Yaskawa INFORM job: SEQUENCE1.JBI

/JOB
//NAME SEQUENCE1
//POS
///NPOS 16,16,16,0,0,0
///TOOL 2
///POSTYPE PULSE
///PULSE
C00000=-123787,24304,7596,24730,-10033,18005
C00001=-124139,38523,-23923,25034,13017,13567
C00002=-125998,37166,-27833,25904,14956,13586
C00003=-126763,36701,-29332,26274,15729,13590
C00004=-125268,29724,-35802,30017,19497,16175
C00005=-123323,21362,-43824,35562,24187,18403
C00006=-122752,14684,-49649,39024,28143,20530
C00007=-122789,12113,-51767,40794,30645,22351
C00008=-122154,60097,-5285,37527,25638,24249
C00009=-122371,55552,-10496,40477,30561,26040
C00010=-122762,52079,-14356,42105,33589,27254
C00011=-124409,44094,-22923,44998,40650,30262
C00012=-126075,39257,-28036,46274,45650,32666
C00013=-125315,37235,-28983,45882,45162,32673
C00014=-123361,32258,-31183,44881,43872,32693
C00015=-122892,16140,-12651,31673,29212,39259
///TOOL 0
BC00000=204858
BC00001=204858
BC00002=204858
BC00003=204858
BC00004=204858
BC00005=204858
BC00006=204858
BC00007=204858
BC00008=204858
BC00009=204858
BC00010=204858
BC00011=204858
BC00012=204858
BC00013=204858
BC00014=204858
BC00015=204858
EC00000=-379617,176269
EC00001=-379617,176269
EC00002=-379617,176269
EC00003=-379617,176269
EC00004=-379617,176269
EC00005=-379617,176269
EC00006=-379617,176269
EC00007=-379617,176269
EC00008=-379617,176269
EC00009=-379617,176269
EC00010=-379617,176269
EC00011=-379617,176269
EC00012=-379617,176269
EC00013=-379617,176269
EC00014=-379617,176269
EC00015=-379617,176269
//INST
///DATE 2026/05/13 10:02
///ATTR SC,RW
///GROUP1 RB1,BS1
///GROUP2 ST1
NOP
'Sequence1
MEMOF
CLEAR MPF
'Path W11
SSFTOF
MOVJ C00000 BC00000 VJ=100.00  +MOVJ EC00000 VJ=100.00
SMOVL C00001 BC00001 V=1000.0  +MOVJ EC00001
SMOVL C00002 BC00002 V=400.0  +MOVJ EC00002
SMOVL C00003 BC00003 V=10.0 PL=0  +MOVJ EC00003
SMOVL C00004 BC00004 V=10.0  +MOVJ EC00004
SMOVL C00005 BC00005 V=10.0  +MOVJ EC00005
SMOVL C00006 BC00006 V=10.0  +MOVJ EC00006
SMOVL C00007 BC00007 V=10.0  +MOVJ EC00007
SMOVL C00008 BC00008 V=10.0  +MOVJ EC00008
SMOVL C00009 BC00009 V=10.0  +MOVJ EC00009
SMOVL C00010 BC00010 V=10.0  +MOVJ EC00010
SMOVL C00011 BC00011 V=10.0  +MOVJ EC00011
SMOVL C00012 BC00012 V=10.0  +MOVJ EC00012
SMOVL C00013 BC00013 V=400.0  +MOVJ EC00013
SMOVL C00014 BC00014 V=1000.0  +MOVJ EC00014
SMOVL C00015 BC00015 V=1000.0  +MOVJ EC00015
'EndPath W11
END
